(* PLC project sample_project, sample_company sample_product 1 *)
(* stored: creationDateTime 2024-07-18T21:30:47, modificationDateTime 2024-07-18T22:03:54 *)

(* Counter in ST language *)
FUNCTION_BLOCK sample_function_block_ST
  VAR_INPUT
    Reset : BOOL;
  END_VAR
  VAR_OUTPUT
    Out : INT;
  END_VAR
  VAR
    Cnt : INT;
  END_VAR
  VAR_OUTPUT
    Cnt_R : REAL;
  END_VAR
  VAR_EXTERNAL CONSTANT
    ResetCounterValue : INT;
  END_VAR

            IF Reset THEN
  Cnt := ResetCounterValue;
ELSE
  Cnt := Cnt + 1;
END_IF;

Out := Cnt;

Cnt_R := INT_TO_REAL(Cnt);
Cnt_R := FACTORIAL(Cnt_R);

          
END_FUNCTION_BLOCK

PROGRAM sample_program
  VAR_INPUT
    Reset : BOOL;
  END_VAR
  VAR_OUTPUT
    Cnt0 : INT;
    Cnt_R : REAL;
  END_VAR
  VAR
    sample_function_block_ST0 : sample_function_block_ST;
  END_VAR

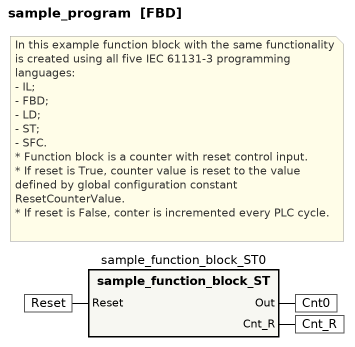
(* FBD diagram, written out as Structured Text *)
(* In this example function block with the same functionality is created using all five IEC 61131-3 programming languages:
- IL;
- FBD;
- LD;
- ST;
- SFC.

* Function block is a counter with reset control input.
* If reset is True, counter value is reset to the value defined by global configuration constant ResetCounterValue.
* If reset is False, conter is incremented every PLC cycle. *)
sample_function_block_ST0(Reset := Reset);
Cnt0 := sample_function_block_ST0.Out;
Cnt_R := sample_function_block_ST0.Cnt_R;
END_PROGRAM

CONFIGURATION sample_config
  VAR_GLOBAL CONSTANT
    ResetCounterValue : INT := 17;
  END_VAR
  RESOURCE sample_resource ON PLC
    TASK sample_task(INTERVAL := T#200ms, PRIORITY := 0);
    PROGRAM sample_task_instance WITH sample_task : sample_program;
  END_RESOURCE
END_CONFIGURATION
